PROGRAM MAIN
VAR
END_VAR

A_Program();

END_PROGRAM

(* stored: Version 1.1.0.1, ProductVersion 3.1.4025.12
   POU MAIN: Id {bbcb6aa6-9912-4447-8c6e-014a2a63340c}, SpecialFunc None *)
